{attribute 'qualified_only'}
{attribute 'strict'}
TYPE E_StateSortingAutoAxis :
(
	WaitForCylinderAtWorkPos 			:= 0,
	MoveAxis,
	StopAxis
);
END_TYPE

(* stored: Version 1.1.0.1, ProductVersion 3.1.4024.15
   DUT E_StateSortingAutoAxis: Id {060bb3ee-0b8b-4f7c-b977-55d41f4dfc73} *)
